TYPE ST_EventMessageParams :
STRUCT	
  Severity : TcEventSeverity;
  Message : T_MessageString;
  Source : T_MaxString;
END_STRUCT
END_TYPE

(* stored: Version 1.1.0.1, ProductVersion 3.1.4024.12
   DUT ST_EventMessageParams: Id {304026b0-5580-06d2-2170-3ee00f189613} *)
